// TwinCAT 3 PLC project PLCData
// ProgramVersion: 3.1.4026.22
// libraries:
//   Tc2_Standard, * (Beckhoff Automation GmbH)
//   Tc2_System, * (Beckhoff Automation GmbH)
//   Tc2_Utilities, * (Beckhoff Automation GmbH)
//   Tc3_IotBase, * (Beckhoff Automation GmbH)
//   Tc3_JsonXml, * (Beckhoff Automation GmbH)
// project tree:
//   DUTs/ DataStruct.TcDUT, DUT_Message.TcDUT
//   / PlcTask.TcTTO
//   POUs/ MAIN.TcPOU (not stored), TO_JSON.TcPOU (not stored)
// real-time tasks:
//   TASK PlcTask: cycle T#10ms, priority 20, ADS port 350
// I/O:
//   DEVICE Device 1 (OPC UA RT), AmsNetId 10.10.11.1.2.1

CONFIGURATION PLCData
    RESOURCE PLC ON TwinCAT3
        TASK PlcTask(INTERVAL := T#10ms, PRIORITY := 20);
        PROGRAM MAIN WITH PlcTask : MAIN;
    END_RESOURCE
END_CONFIGURATION

// ---- DUTs/DataStruct.TcDUT
TYPE DataStruct :
STRUCT
	bTest	: BOOL;
	nTest	: DINT;
	fTest	: LREAL;
	sTest	: STRING;
END_STRUCT
END_TYPE

// ---- DUTs/DUT_Message.TcDUT
TYPE DUT_Message :
STRUCT
	Id	: DINT;
	Message	: STRING(255);
END_STRUCT
END_TYPE
